# B&R Automation Studio project A_FullProject
Automation Studio 4.9

## Configuration Config1

CPU X20CP1686X, AutomationRuntime M4.93, Build 4.1.2, Safety 0.0, Vc V4.73.2

### Task classes (Cpu.sw)
```
Cyclic#4:
  Axis <- Vision.Axis.prg
  Vi_main <- Vision.Vi_main.prg
  Vi_image <- Vision.Vi_image.prg
DataObjects: McAcpSys
NcDataObjects: mcdrivelog
Binaries: arsvcreg, FWRules, McAcpSim, mvLoader, mCoWebSc, visionUnit, McAcpDrv, TCData, udbdef, arflatprv, arcoal, iomap, asfw, Settings, Role, SettingsVC, Config_1, VAMatch, arconfig, VCMyCam, ashwd, sysconf, User, ashwac
Libraries: McBase, MpBase, ViBase, AsZip, FileIO, AsARCfg, powerlnk, AsEPL, AsIO, AsTCP, sys_lib, DataObj, astime, runtime, CoTrace, MpAxis, McAxis, McAcpAx, arssl, asieccon
```

### Hardware
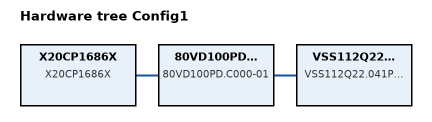
```
80VD100PD.C000-01 : 80VD100PD.C000-01 v2.5.0.0  [PLK1 -> X20CP1686X.IF3 (NodeNumber=1) [Cable Type=PowerlinkCable, Length=10, Version=1.0.0.3]; PLK2 -> VSS112Q22.041P-000.PLK1 (NodeNumber=1) [Cable Type=PowerlinkCable, Length=10, Version=1.0.0.3]]
  DriveConfiguration/Module:
    McAcoposTypeID = AcoposMicroDConfig
    ActivateACOPOSSimulationOnPLC = 0
  DriveConfiguration/Channel[1]/RealAxis:
    AxisReference = 
    MechanicalElementsIsInvisible = 0
  DriveConfiguration/Channel[1]/RealAxis/MechanicalElements/Gearbox:
    InputIsReadOnly = 0
    Input = 1
    OutputIsReadOnly = 0
    Output = 1
  DriveConfiguration/Channel[1]/RealAxis/MechanicalElements/RotaryToLinearTransformation:
    ReferenceDistanceIsReadOnly = 0
    ReferenceDistance = 1
  DriveConfiguration/Channel[1]/RealAxis/Controller:
    ModeIsReadOnly = 0
    Mode = PositionController
  DriveConfiguration/Channel[1]/RealAxis/Controller/Mode/Position:
    ProportionalGain = 200
    IntegrationTime = 0.0
    PredictionTime = 0.0004
    TotalDelayTime = 0.0004
  DriveConfiguration/Channel[1]/RealAxis/Controller/Mode/Speed:
    ProportionalGainIsReadOnly = 0
    ProportionalGain = 0.9
    IntegrationTimeIsReadOnly = 0
    IntegrationTime = 0.0
    FilterTimeIsReadOnly = 0
    FilterTime = 0.0
  DriveConfiguration/Channel[1]/RealAxis/Controller/Mode/LoopFilters:
    LoopFilterXIsReadOnly = 0
    LoopFilter1 = NotUsed
    LoopFilter2 = NotUsed
    LoopFilter3 = NotUsed
  DriveConfiguration/Channel[1]/RealAxis/Homing:
    ModeIsReadOnly = 0
    Mode = Direct
  DriveConfiguration/Channel[1]/RealAxis/Homing/Mode:
    Position = 0.0
    ReferencePulse = NotUsed
  DriveConfiguration/Channel[1]/RealAxis/Homing:
    RestorePositionVariable = 
  DriveConfiguration/Channel[1]/RealAxis/StopReaction:
    QuickstopIsReadOnly = 0
    Quickstop = DecelerationLimit
    DriveErrorIsReadOnly = 0
    DriveError = DecelerationLimit
  DriveConfiguration/Channel[1]/RealAxis/MovementErrorLimits:
    PositionError = 1.0
    VelocityErrorMonitoring = Automatic1
  DriveConfiguration/Channel[1]/RealAxis:
    JerkFilterIsReadOnly = 0
    JerkFilter = NotUsed
    ZeroVibrationFilter = NotUsed
  DriveConfiguration/Channel[1]/RealAxis/DigitalInputs/HomingSwitch:
    SourceIsReadOnly = 0
    Source = NotUsed
    Level = High
  DriveConfiguration/Channel[1]/RealAxis/DigitalInputs/PositiveLimitSwitch:
    SourceIsReadOnly = 0
    Source = NotUsed
    Level = High
  DriveConfiguration/Channel[1]/RealAxis/DigitalInputs/NegativeLimitSwitch:
    SourceIsReadOnly = 0
    Source = NotUsed
    Level = High
  DriveConfiguration/Channel[1]/RealAxis/DigitalInputs/Trigger1:
    Source = X2Trigger1
    Level = High
  DriveConfiguration/Channel[1]/RealAxis/DigitalInputs/Trigger2:
    Source = X2Trigger2
    Level = High
  DriveConfiguration/Channel[1]/RealAxis/DigitalInputs/Quickstop:
    Input = Trigger2
  DriveConfiguration/Channel[1]/RealAxis/Simulation:
    SimulationModeOnPLC = SetValueGeneration
    SimulationModeOnACOPOS = NotUsed
  DriveConfiguration/Channel[1]:
    ExternalEncoderAxis = NotUsed
  DriveConfiguration/Channel[2]/RealAxis:
    AxisReference = gAxis_1
    MechanicalElementsIsInvisible = 0
  DriveConfiguration/Channel[2]/RealAxis/MechanicalElements/Gearbox:
    InputIsReadOnly = 0
    Input = 1
    OutputIsReadOnly = 0
    Output = 1
  DriveConfiguration/Channel[2]/RealAxis/MechanicalElements/RotaryToLinearTransformation:
    ReferenceDistanceIsReadOnly = 0
    ReferenceDistance = 1
  DriveConfiguration/Channel[2]/RealAxis/Controller:
    ModeIsReadOnly = 0
    Mode = PositionController
  DriveConfiguration/Channel[2]/RealAxis/Controller/Mode/Position:
    ProportionalGain = 200
    IntegrationTime = 0.0
    PredictionTime = 0.0004
    TotalDelayTime = 0.0004
  DriveConfiguration/Channel[2]/RealAxis/Controller/Mode/Speed:
    ProportionalGainIsReadOnly = 0
    ProportionalGain = 0.9
    IntegrationTimeIsReadOnly = 0
    IntegrationTime = 0.0
    FilterTimeIsReadOnly = 0
    FilterTime = 0.0
  DriveConfiguration/Channel[2]/RealAxis/Controller/Mode/LoopFilters:
    LoopFilterXIsReadOnly = 0
    LoopFilter1 = NotUsed
    LoopFilter2 = NotUsed
    LoopFilter3 = NotUsed
  DriveConfiguration/Channel[2]/RealAxis/Homing:
    ModeIsReadOnly = 0
    Mode = Direct
  DriveConfiguration/Channel[2]/RealAxis/Homing/Mode:
    Position = 0.0
    ReferencePulse = NotUsed
  DriveConfiguration/Channel[2]/RealAxis/Homing:
    RestorePositionVariable = 
  DriveConfiguration/Channel[2]/RealAxis/StopReaction:
    QuickstopIsReadOnly = 0
    Quickstop = DecelerationLimit
    DriveErrorIsReadOnly = 0
    DriveError = DecelerationLimit
  DriveConfiguration/Channel[2]/RealAxis/MovementErrorLimits:
    PositionError = 1.0
    VelocityErrorMonitoring = Automatic1
  DriveConfiguration/Channel[2]/RealAxis:
    JerkFilterIsReadOnly = 0
    JerkFilter = NotUsed
    ZeroVibrationFilter = NotUsed
  DriveConfiguration/Channel[2]/RealAxis/DigitalInputs/HomingSwitch:
    SourceIsReadOnly = 0
    Source = NotUsed
    Level = High
  DriveConfiguration/Channel[2]/RealAxis/DigitalInputs/PositiveLimitSwitch:
    SourceIsReadOnly = 0
    Source = NotUsed
    Level = High
  DriveConfiguration/Channel[2]/RealAxis/DigitalInputs/NegativeLimitSwitch:
    SourceIsReadOnly = 0
    Source = NotUsed
    Level = High
  DriveConfiguration/Channel[2]/RealAxis/DigitalInputs/Trigger1:
    Source = X2Trigger1
    Level = High
  DriveConfiguration/Channel[2]/RealAxis/DigitalInputs/Trigger2:
    Source = X2Trigger2
    Level = High
  DriveConfiguration/Channel[2]/RealAxis/DigitalInputs/Quickstop:
    Input = Trigger2
  DriveConfiguration/Channel[2]/RealAxis/Simulation:
    SimulationModeOnPLC = SetValueGeneration
    SimulationModeOnACOPOS = NotUsed
  DriveConfiguration/Channel[2]:
    ExternalEncoderAxis = NotUsed
VSS112Q22.041P-000 : VSS112Q22.041P-000 v1.11.0.922  [PLK1 -> 80VD100PD.C000-01.PLK2 (NodeNumber=2) [Cable Type=PowerlinkCable, Length=10, Version=1.0.0.3]]
  Supervision = off
  VisionConfig = VCMyCam
X20CP1686X : X20CP1686X v1.8.2.0
  Connector IF2:
    ActivateDevice = 1
    Mode = Manual
    InternetAddress = 192.168.1.100
    SubnetMask = 255.255.255.0
    ActivateSnmp = 2
  Connector IF3:
    MtuSize = 1500
    InternetAddress = 192.168.200.240
    SubnetMask = 255.255.255.0
  ConfigurationID = VisionSample_AxisSync_Config1
  UserPartitionSize = 500
  TimerDeviceType = EPLX2X
  TimerDevice = X20CP1686X.IF3
  FileDevice1
  FileDeviceName1 = CF
  FileDevicePath1 = F:\
  FtpUser1
  FtpUsername1 = test
  FtpUserPassword1 = QkT+VSyJDE68GyHqQqfzGbDLRHfoQvgBAqgTYwFwErQ=  // test
  FtpUserSalt1 = 9xieoJwW
  FTPAccessRight1 = 0
  FTPdevice1 = ALL
  ActivateOpcUa = 1
  OpcUaInformationModels_PV_Version = 1
```

### IoMap.iom - X20CP1686X/IoMap.iom
```iecst
VAR_CONFIG
	::Vi_main:VisionCtrl.Parameters.SetFocus AT %QW."VSS112Q22.041P-000".SetFocus;
	::Vi_main:VisionCtrl.Parameters.ExposureTime AT %QD."VSS112Q22.041P-000".ExposureTime01;
	::Vi_main:VisionCtrl.Parameters.FlashColor AT %QB."VSS112Q22.041P-000".FlashColor01;
	::Vi_main:VisionCtrl.Parameters.FlashSegment AT %QB."VSS112Q22.041P-000".FlashSegment01;
	::Vi_main:CompletedAcquisitionCntOld AT %IB."VSS112Q22.041P-000".CompletedAcquisitionCnt;
END_VAR
```

### Config_1.axis - X20CP1686X/mappMotion/Config_1.axis
```
Element gAxis_1 (Type=axis)
  BaseTypeIsReadOnly = 0
  BaseType = RotaryPeriodic
    MeasurementUnitIsReadOnly = 0
    MeasurementUnit = 17476
    MeasurementResolutionIsReadOnly = 0
    MeasurementResolution = 0.01
    CountDirectionIsReadOnly = 0
    CountDirection = Standard
    PeriodSettings:
      Period = 360.0
  MovementLimitsIsReadOnly = 0
  MovementLimits = Internal
    Position:
      LowerLimitMin = -1.79769313486231E308
      UpperLimitMax = 1.79769313486231E308
      LowerLimit = -1000.0
      UpperLimit = 1000.0
    VelocityIsReadOnly = 0
    Velocity:
      VelocityMax = 3.4E38
      Velocity = 6000
    AccelerationIsReadOnly = 0
    Acceleration:
      AccelerationMax = 3.4E38
      Acceleration = 36000
    DecelerationIsReadOnly = 0
    Deceleration:
      DecelerationMax = 3.4E38
      Deceleration = 36000
  Alarms = None
```

### SettingsVC.vicfg - X20CP1686X/mappVision/SettingsVC.vicfg
```
Element VisionSettings (Type=vicfg)
  ActivateVisualization = TRUE
  FileDeviceName
  Permissions:
    WriteAccessRole = Everyone
  DeepLearning:
    CustomDlNetworks:
      DLFileDeviceName
      DLNetworkBuildPath
```

### VCMyCam.visioncomponent - X20CP1686X/mappVision/VCMyCam.visioncomponent
```
Element VCMyCam (Type=visioncomponent)
  VisionApplicationReference = VAMatch
```

## Logical view

Binary libraries used (declarations not repeated): brsystem, McAcpAx 5.28.2, McBase 5.28.2, powerlnk, ViBase 5.28.1

### Package Logical/Libraries - Globale Bibliotheken

### MpAxisCfg.typ
```iecst
TYPE
	MpAXBAxBaseTypEnum :
		( (*Axis base type*)
		mcAXB_BASE_TYPE_LIN_BD := 0, (*Linear bounded - Linear axis with bounded movement scope*)
		mcAXB_BASE_TYPE_LIN := 1, (*Linear - Linear axis*)
		mcAXB_BASE_TYPE_LIN_PER := 2, (*Linear periodic - Linear axis with periodic movement scope*)
		mcAXB_BASE_TYPE_ROT_BD := 10, (*Rotary bounded - Rotary axis with bounded movement scope*)
		mcAXB_BASE_TYPE_ROT := 11, (*Rotary - Rotary axis*)
		mcAXB_BASE_TYPE_ROT_PER := 12 (*Rotary periodic - Rotary axis with periodic movement scope*)
		);
	MpAXBAxMeasUnitEnum :
		( (*Measurement unit for the axis*)
		mcAXB_MEAS_UNIT_G_SET := 0, (*Global settings*)
		mcAXB_MEAS_UNIT_MILIMETERS := 5066068, (*Milimeters*)
		mcAXB_MEAS_UNIT_M := 5067858, (*Meters*)
		mcAXB_MEAS_UNIT_INCH := 4804168, (*Inches*)
		mcAXB_MEAS_UNIT_DEG := 17476, (*Degrees*)
		mcAXB_MEAS_UNIT_GRAD := 4274481, (*Gradians*)
		mcAXB_MEAS_UNIT_REV := 5059636, (*Revolutions*)
		mcAXB_MEAS_UNIT_GEN := -1 (*Generic*)
		);
	MpAXBAxCntDirEnum :
		( (*Direction of the axis in which the position value is increasing*)
		mcAXB_COUNT_DIR_STD := 0, (*Standard*)
		mcAXB_COUNT_DIR_INV := 1 (*Inverse*)
		);
	MpAXBAxMoveLimTypEnum :
		( (*Movement limits settings*)
		mcAXB_MOV_LIM_STD := 0, (*Standard*)
		mcAXB_MOV_LIM_PATH_CTRL_AX := 1, (*Path controlled axis*)
		mcAXB_MOV_LIM_LIM_SET_REF := 2 (*Limit set reference*)
		);
	MpAXBAxMoveLimPosType : STRUCT (*Movement range of the axis via two position boundaries; Only for bounded axis*)
		LowerLimit : LREAL; (*Lower software limit position [Measurement units]*)
		UpperLimit : LREAL; (*Upper software limit position [Measurement units]*)
	END_STRUCT;
	MpAXBAxMoveLimVelType : STRUCT (*Limits for the velocity of the axis*)
		Positive : REAL; (*Velocity limit in positive movement direction [Measurement units/s]*)
		Negative : REAL; (*Velocity limit in negative movement direction [Measurement units/s]*)
	END_STRUCT;
	MpAXBAxMoveLimType : STRUCT
		Type : MpAXBAxMoveLimTypEnum; (*Movement limits settings*)
		Position : MpAXBAxMoveLimPosType; (*Movement range of the axis via two position boundaries; Only for bounded axis*)
		Velocity : MpAXBAxMoveLimVelType; (*Limits for the velocity of the axis*)
		Acceleration : REAL; (*Acceleration limit in any movement direction [Measurement units/s²]*)
		Deceleration : REAL; (*Deceleration limit in any movement direction [Measurement units/s²]*)
		Jerk : REAL; (*Jerk limit in any movement direction [Measurement units/s³]; Only for [Measurement units/s³]*)
		Torque : REAL; (*Torque limit in any movement direction; Only for Axis of type rotary; only for limits type internal path controlled [Nm]*)
		Force : REAL; (*Force limit in any movement direction [N]; Only for Axis of type linear; only for limits type internal path controlled [N]*)
		LimitSetReference : STRING[250]; (*Name of the limit reference; only for limits type external*)
	END_STRUCT;
	MpAXBAxType : STRUCT (*Axis configuration*)
		BaseType : MpAXBAxBaseTypEnum; (*Axis base type*)
		MeasurementUnit : MpAXBAxMeasUnitEnum; (*Measurement unit for the axis*)
		MeasurementResolution : LREAL; (*Possible resolution of measurement unit that can be achieved [Measurement resolution]*)
		CountDirection : MpAXBAxCntDirEnum; (*Direction of the axis in which the position value is increasing*)
		Period : LREAL; (*The value range for axis positions is [0 , Period]; Only for Axis of type periodic [Measurement units]*)
		MovementLimits : MpAXBAxMoveLimType;
	END_STRUCT;
	MpAXBDrvMechElmGBType : STRUCT
		Input : DINT; (*Number of rotations on the encoder side [Revolutions] [Revolutions]*)
		Output : DINT; (*Number of rotations on the load side which correspond to the number of rotations onthe encoder side [Revolutions] [Revolutions]*)
	END_STRUCT;
	MpAXBDrvMechElmRotToLinTrfType : STRUCT (*Specifies a transformation factor between the output of the gear and the actual load movement*)
		ReferenceDistance : LREAL; (*Reference distance which is considered for an axis positioning [Measurement units/Gearbox output revolution] [Measurement units/Gearbox output revolution]*)
	END_STRUCT;
	MpAXBDrvMechElmType : STRUCT (*Parameter of hardware elements situated between motor encoder and load which influence the scaling*)
		Gearbox : MpAXBDrvMechElmGBType;
		RotaryToLinearTransformation : MpAXBDrvMechElmRotToLinTrfType; (*Specifies a transformation factor between the output of the gear and the actual load movement*)
	END_STRUCT;
	MpAXBDrvCtrlModEnum :
		( (*Mode of the axis controller*)
		mcAXB_CTRL_MODE_POS := 0, (*Position - Automatic speed feed-forward with prediction time > 0*)
		mcAXB_CTRL_MODE_POS_W_TORQ_FF := 1, (*Position with torque FF - Torque feed-forward with specified parameters*)
		mcAXB_CTRL_MODE_POS_MDL_BASED := 3, (*Position model based - Model based control with specified parameters*)
		mcAXB_CTRL_MODE_V_FREQ := 2, (*Voltage frequency - Voltage/frequency control of induction motor with specified parameters*)
		mcAXB_CTRL_MODE_STP_CUR := 4, (*Stepper current - StpAx only. Current controller is used*)
		mcAXB_CTRL_MODE_STP_POS_AND_CUR := 5, (*Stepper position and current - StpAx only. Position and current controller are used*)
		mcAXB_CTRL_MODE_NOT_USE := 6 (*Not used - Controller not used*)
		);
	MpAXBDrvCtrlPosType : STRUCT (*Position controller parameters*)
		ProportionalGain : REAL; (*Proportional amplification [1/s]*)
		IntegrationTime : REAL; (*Integral action time [s]*)
		TotalDelayTime : REAL; (*Total delay time [s]*)
		PredictionTime : REAL; (*Prediction time [s]*)
		MaximumProportionalAction : REAL; (*Maximum proportional action. Only for StpAx and PureVax with GPAI [Measurement units/s]*)
		MaximumIntegralAction : REAL; (*Maximum integral action. Only for PureVax with GPAI [Measurement units/s]*)
	END_STRUCT;
	MpAXBDrvCtrlSpdType : STRUCT (*Speed controller parameters*)
		ProportionalGain : REAL; (*Proportional amplification [1/s]*)
		IntegrationTime : REAL; (*Integral action time [s]*)
		FilterTime : REAL; (*Filter time constant [s]*)
	END_STRUCT;
	MpAXBDrvCtrlFFwdModEnum :
		( (*Mode of the axis controller*)
		mcAXB_FF_MODE_STD := 0, (*Standard*)
		mcAXB_FF_MODE_PRED_SPD := 1, (*Predictive speed*)
		mcAXB_FF_MODE_TWO_MASS_MDL := 2 (*Two mass model*)
		);
	MpAXBDrvCtrlFFwdType : STRUCT (*Torque feed-forward control parameters*)
		Mode : MpAXBDrvCtrlFFwdModEnum; (*Mode of the axis controller*)
		TorqueLoad : REAL; (*Load torque [Nm]*)
		TorquePositive : REAL; (*Torque in positive direction [Nm]*)
		TorqueNegative : REAL; (*Torque in negative direction [Nm]*)
		SpeedTorqueFactor : REAL; (*Speed torque factor [Nms]*)
		Inertia : REAL; (*Mass moment of inertia [kgm²]*)
		AccelerationFilterTime : REAL; (*Acceleration filter time constant [s]*)
		PredictionTime : REAL; (*Prediction time [s]*)
	END_STRUCT;
	MpAXBDrvCtrlFdbkModEnum :
		( (*Mode of the axis controller*)
		mcAXB_CTLR_FEED_STD := 0, (*Standard*)
		mcAXB_CTLR_FEED_ONE_MASS_MDL := 1, (*One mass model*)
		mcAXB_CTLR_FEED_TWO_MASS_MDL := 2, (*Two mass model*)
		mcAXB_CTLR_FEED_TWO_ENC_SPD := 3 (*Two encoder speed*)
		);
	MpAXBDrvCtrlFdbkType : STRUCT (*Feedback control parameters*)
		Mode : MpAXBDrvCtrlFdbkModEnum; (*Mode of the axis controller*)
		SpeedMixingFactor : REAL; (*Load torque [Nm]*)
		SpeedProportionalGain : REAL; (*Torque in positive direction [Nm]*)
	END_STRUCT;
	MpAXBDrvCtrlMdlMass1Type : STRUCT (*Mass 1 parameters*)
		Inertia : REAL; (*Mass moment of inertia [kgm²]*)
		ViscousFriction : REAL; (*Viscous friction [Nms]*)
	END_STRUCT;
	MpAXBDrvCtrlMdlMass2Type : STRUCT (*Mass 2 parameters*)
		Inertia : REAL; (*Mass moment of inertia [kgm²]*)
		ViscousFriction : REAL; (*Viscous friction [Nms]*)
		Stiffness : REAL; (*Stiffness of the coupling to mass 1 [Nm/rad]*)
		Damping : REAL; (*Damping of the coupling to mass 1 [Nms/rad]*)
	END_STRUCT;
	MpAXBDrvCtrlMdlType : STRUCT (*Load model parameters*)
		Mass1 : MpAXBDrvCtrlMdlMass1Type; (*Mass 1 parameters*)
		Mass2 : MpAXBDrvCtrlMdlMass2Type; (*Mass 2 parameters*)
	END_STRUCT;
	MpAXBDrvCtrlVFreqCtrlTypEnum :
		( (*Type of characteristic curve*)
		mcAXB_VF_TYP_LIN := 129, (*Linear - Linear characteristic curve*)
		mcAXB_VF_TYP_CONST_LD_TORQ := 131, (*Constant load torque - Characteristic curve for quadratic load curves*)
		mcAXB_VF_TYP_QUAD := 130 (*Quadratic - Characteristic curve for quadratic load curves*)
		);
	MpAXBDrvCtrlVFreqCtrlAutCfgEnum :
		( (*Automatic configuration of parameters*)
		mcAXB_VF_AUTO_CFG_NOT_USE := 0, (*Not used*)
		mcAXB_VF_AUTO_CFG_MOT_PAR_BASED := 1 (*Motor parameter based*)
		);
	MpAXBDrvCtrlVFreqCtrlType : STRUCT (*V/f control parameters*)
		Type : MpAXBDrvCtrlVFreqCtrlTypEnum; (*Type of characteristic curve*)
		AutomaticConfiguration : MpAXBDrvCtrlVFreqCtrlAutCfgEnum; (*Automatic configuration of parameters*)
		SlipCompensation : REAL; (*Slip compensation: Multiplication factor of compensated frequency*)
		TotalDelayTime : REAL; (*Total delay time [s]*)
		BoostVoltage : REAL; (*Boost voltage [V]*)
		RatedVoltage : REAL; (*Rated voltage [V]*)
		RatedFrequency : REAL; (*Rated frequency [cps]*)
	END_STRUCT;
	MpAXBDrvCtrlLoopFltrTypEnum :
		( (*Type of the loop filter*)
		mcAXB_LP_FLTR_NOT_USE := 0, (*Not used - Filter is not active*)
		mcAXB_LP_FLTR_LOW_PASS_2ND_ORD := 1, (*Low pass 2nd order*)
		mcAXB_LP_FLTR_NOTCH := 2, (*Notch*)
		mcAXB_LP_FLTR_BIQUAD := 3, (*Biquad*)
		mcAXB_LP_FLTR_DISC_TIME_TRAN_FUN := 4, (*Discrete time transfer function*)
		mcAXB_LP_FLTR_LIM := 5, (*Limiter*)
		mcAXB_LP_FLTR_LIN_LIM := 6, (*Linear limitation*)
		mcAXB_LP_FLTR_RISE_TIME_LIM := 7, (*Rise time limitation*)
		mcAXB_LP_FLTR_COMP := 8 (*Compensation*)
		);
	MpAXBLoopFltrLP2ndOrdType : STRUCT (*Lowpass 2nd order*)
		CutOffFrequency : REAL; (*Cut off frequency [Hz]*)
	END_STRUCT;
	MpAXBLoopFltrNotchType : STRUCT (*Notch*)
		CenterFrequency : REAL; (*Center frequency [Hz]*)
		Bandwidth : REAL; (*Bandwidth [Hz]*)
	END_STRUCT;
	MpAXBLoopFltrBiquadType : STRUCT (*Biquad*)
		FrequencyNumerator : REAL; (*Frequency numerator [Hz]*)
		DampingNumerator : REAL; (*Damping numerator*)
		FrequencyDenominator : REAL; (*Frequency denominator [Hz]*)
		DampingDenominator : REAL; (*Damping Denominator*)
	END_STRUCT;
	MpAXBLoopFltrDiscTimeTranFunType : STRUCT (*Discrete time transfer function*)
		CoeffA0DenominatorPolynomial : REAL; (*Coefficient a0 of denominator polynomial*)
		CoeffA1DenominatorPolynomial : REAL; (*Coefficient a1 of denominator polynomial*)
		CoeffB0NominatorPolynomial : REAL; (*Coefficient b0 of numerator polynomial*)
		CoeffB1NominatorPolynomial : REAL; (*Coefficient b1 of numerator polynomial*)
		CoeffB2NominatorPolynomial : REAL; (*Coefficient b2 of numerator polynomial*)
	END_STRUCT;
	MpAXBLoopFltrLimLimTypEnum :
		( (*Select if for the limit a fixed value or if the value of an ACOPOS ParID is used*)
		mcAXB_LOOP_FLTR_LIM_TYPE_PARID := 0, (*ParId*)
		mcAXB_LOOP_FLTR_LIM_TYPE_FIX_VAL := 1 (*Fixed value*)
		);
	MpAXBLoopFltrLimLimType : STRUCT (*Positive limit setting*)
		Type : MpAXBLoopFltrLimLimTypEnum; (*Select if for the limit a fixed value or if the value of an ACOPOS ParID is used*)
		ParID : UINT; (*ParID*)
		Value : REAL; (*Value [A]*)
	END_STRUCT;
	MpAXBLoopFltrLimType : STRUCT (*Limiter*)
		PositiveLimit : MpAXBLoopFltrLimLimType; (*Positive limit setting*)
		NegativeLimit : MpAXBLoopFltrLimLimType; (*Negative limit setting*)
	END_STRUCT;
	MpAXBLoopFltrLinLimType : STRUCT (*Linear limitation*)
		InputParID : UINT; (*ACOPOS ParID for the input*)
		InputLimit : REAL; (*Input limit value for full limitation*)
		Gradient : REAL; (*Gradient*)
	END_STRUCT;
	MpAXBLoopFltrRiseTimeLimType : STRUCT (*Rise time limitation*)
		RiseTime : REAL; (*Rise time [s]*)
		NormalizedLimit : REAL; (*Normalized limit*)
	END_STRUCT;
	MpAXBLoopFltrCompType : STRUCT (*Compensation*)
		MultiplicationFactorParID : UINT; (*Multiplication Factor ParID*)
		AdditiveValueParID : UINT; (*Additive Value ParID*)
	END_STRUCT;
	MpAXBDrvCtrlLoopFltrLoopFltrType : STRUCT (*Type of the loop filter*)
		Type : MpAXBDrvCtrlLoopFltrTypEnum; (*Type of the loop filter*)
		Lowpass2ndOrder : MpAXBLoopFltrLP2ndOrdType; (*Lowpass 2nd order*)
		Notch : MpAXBLoopFltrNotchType; (*Notch*)
		Biquad : MpAXBLoopFltrBiquadType; (*Biquad*)
		DiscreteTimeTransferFunction : MpAXBLoopFltrDiscTimeTranFunType; (*Discrete time transfer function*)
		Limiter : MpAXBLoopFltrLimType; (*Limiter*)
		LinearLimitation : MpAXBLoopFltrLinLimType; (*Linear limitation*)
		RiseTimeLimitation : MpAXBLoopFltrRiseTimeLimType; (*Rise time limitation*)
		Compensation : MpAXBLoopFltrCompType; (*Compensation*)
	END_STRUCT;
	MpAXBDrvCtrlLoopFltrType : STRUCT (*Parameters of the loop filters*)
		LoopFilter : ARRAY[0..2] OF MpAXBDrvCtrlLoopFltrLoopFltrType; (*Type of the loop filter*)
	END_STRUCT;
	MpAXBDrvCtrlCurModEnum :
		( (*Mode of current controller*)
		mcAXB_CUR_CTRL_MODE_STD := 0 (*Standard*)
		);
	MpAXBDrvCtrlCurType : STRUCT (*Current controller parameters; Only for stepper axis*)
		Mode : MpAXBDrvCtrlCurModEnum; (*Mode of current controller*)
		StandstillCurrent : REAL; (*Current that is used when no movement is active [A]*)
		ConstantSpeedCurrent : REAL; (*Current that is used when a movement with a constant speed is active [A]*)
		SpeedChangeCurrent : REAL; (*Current that is used when the axis is accelerating or decelerating [A]*)
		FullStepThreshold : REAL; (*Speed of the motor where the driver switch from microstep to full step mode [rpm]*)
		MotorSettlingTime : REAL; (*Minimum time between when the motor is powered on to when the DrvOk bit is set. Settings made in steps of 10 ms. [s]*)
		DelayedCurrentSwitchOff : REAL; (*Time for a delayed motor switch off after it is decelerated to zero because of a settime fault. Setting is made in steps of 100 ms. [s]*)
	END_STRUCT;
	MpAXBDrvCtrlType : STRUCT (*Axis controller parameters*)
		Mode : MpAXBDrvCtrlModEnum; (*Mode of the axis controller*)
		Position : MpAXBDrvCtrlPosType; (*Position controller parameters*)
		Speed : MpAXBDrvCtrlSpdType; (*Speed controller parameters*)
		FeedForward : MpAXBDrvCtrlFFwdType; (*Torque feed-forward control parameters*)
		Feedback : MpAXBDrvCtrlFdbkType; (*Feedback control parameters*)
		Model : MpAXBDrvCtrlMdlType; (*Load model parameters*)
		VoltageFrequencyControl : MpAXBDrvCtrlVFreqCtrlType; (*V/f control parameters*)
		LoopFilters : MpAXBDrvCtrlLoopFltrType; (*Parameters of the loop filters*)
		Current : MpAXBDrvCtrlCurType; (*Current controller parameters; Only for stepper axis*)
	END_STRUCT;
	MpAXBDrvHomeType : STRUCT (*Homing mode and parameters which can be used within the application program as pre-configured setting*)
		Mode : McHomingModeEnum; (*Mode of the axis controller*)
		Position : LREAL; (*Home position [Measurement units]*)
		ReferencePulse : McSwitchEnum; (*Use reference pulse of encoder*)
		ReferencePulseBlockingDistance : LREAL; (*Distance for blocking the activation of triggering reference pulse [Measurement units]*)
		StartVelocity : REAL; (*Speed for searching the reference switch [Measurement units/s]*)
		HomingVelocity : REAL; (*Speed which is used while searching for the homing event (e.g. after reference switch has been reached) [Measurement units/s]*)
		Acceleration : REAL; (*Acceleration for homing movement [Measurement units/s²]*)
		SwitchEdge : McDirectionEnum; (*Edge of reference switch*)
		HomingDirection : McDirectionEnum; (*Movement direction in which the homing event is evaluated*)
		StartDirection : McDirectionEnum; (*Start direction of movement for searching the reference*)
		KeepDirection : McSwitchEnum; (*Keep direction (move only in one direction)*)
		TorqueLimit : REAL; (*Torque limit for homing on block [Nm]*)
		PositionErrorStopLimit : LREAL; (*Lag error for stop of the homing movement [Measurement units/s²]*)
		BlockDetectionPositionError : LREAL; (*Lag error for block detection [Measurement units]*)
		RestorePositionVariable : STRING[250]; (*Remanent variable used for homing mode: Restore position*)
	END_STRUCT;
	MpAXBDrvStopReacQstopEnum :
		( (*Reaction in case of a quickstop which is caused by an active quickstop input*)
		mcAXB_QSTOP_RCT_DEC_LIM := 0, (*Deceleration limit*)
		mcAXB_QSTOP_RCT_DEC_LIM_W_JERK := 1, (*Deceleration limit with jerk*)
		mcAXB_QSTOP_RCT_TORQ_LIM := 2, (*Torque limit*)
		mcAXB_QSTOP_RCT_INDUCT_HALT := 3 (*Induction halt*)
		);
	MpAXBDrvStopReacDrvErrEnum :
		( (*Reaction in case of an error stop which is caused by a drive error*)
		mcAXB_ERR_RCT_DEC_LIM := 0, (*Deceleration limit*)
		mcAXB_ERR_RCT_INDUCT_HALT := 1, (*Induction halt*)
		mcAXB_ERR_RCT_COAST_STANDSTILL := 2, (*Coast standstill*)
		mcAXB_ERR_RCT_CYC_DEC_AXESGROUP := 3 (*Cyclic deceleration AxesGroup*)
		);
	MpAXBDrvStopReacType : STRUCT (*Reactions of the axis in case of certain stop conditions*)
		Quickstop : MpAXBDrvStopReacQstopEnum; (*Reaction in case of a quickstop which is caused by an active quickstop input*)
		DriveError : MpAXBDrvStopReacDrvErrEnum; (*Reaction in case of an error stop which is caused by a drive error*)
	END_STRUCT;
	MpAXBDrvMovVelErrMonEnum :
		( (*Velocity error monitoring mode*)
		mcAXB_VEL_MON_AUT_1 := 0, (*Automatic 1*)
		mcAXB_VEL_MON_AUT_2 := 1, (*Automatic 2*)
		mcAXB_VEL_MON_USR_DEF := 2, (*User defined*)
		mcAXB_VEL_MON_NOT_USE := 3 (*Not used*)
		);
	MpAXBDrvMovementErrorLimitsType : STRUCT (*Limit values that result in a stop reaction when exceeded*)
		PositionError : LREAL; (*Lag error limit for stopping a movement [Measurement units]*)
		VelocityErrorMonitoring : MpAXBDrvMovVelErrMonEnum; (*Velocity error monitoring mode*)
		VelocityError : REAL; (*Velocity error limit for stopping a movement [Measurement units/s]*)
	END_STRUCT;
	MpAXBDrvJerkFilterTypEnum :
		( (*Jerk filter setting*)
		mcAXB_JERK_FLTR_NOT_USE := 0, (*Not used*)
		mcAXB_JERK_FLTR_TIME := 1, (*Time*)
		mcAXB_JERK_FLTR_LIM := 2 (*Limited*)
		);
	MpAXBDrvJerkFilterType : STRUCT (*Jerk filter*)
		Type : MpAXBDrvJerkFilterTypEnum; (*Jerk filter setting*)
		Jerk : REAL; (*Dependant on selected type it is either the jerk limit in any movement direction or a jerk filter time.*)
	END_STRUCT;
	MpAXBDrvDigInLevelEnum :
		( (*Level of the digital input hardware which leads to an active level of the functionality*)
		mcAXB_DI_LEVEL_HIGH := 0, (*High*)
		mcAXB_DI_LEVEL_LOW := 1 (*Low*)
		);
	MpAXBDrvDigInSrcEnum :
		( (*Source of the digital input which is used for this functionality*)
		mcAXBDI_NOT_USE := 0, (*Not used*)
		mcAXBDI_ACP_DIG_IN_X8TRG_1 := 1, (*ACOPOS digital in X8.Trigger 1*)
		mcAXBDI_ACP_DIG_IN_X8TRG_2 := 2, (*ACOPOS digital in X8.Trigger 2*)
		mcAXBDI_ACP_DIG_IN_SS1X41X1 := 3, (*ACOPOS digital in SS1.X41x.1*)
		mcAXBDI_ACP_DIG_IN_SS1X41X2 := 4, (*ACOPOS digital in SS1.X41x.2*)
		mcAXBDI_ACP_DIG_IN_SS1X41X3 := 5, (*ACOPOS digital in SS1.X41x.3*)
		mcAXBDI_ACP_DIG_IN_SS1X41X4 := 6, (*ACOPOS digital in SS1.X41x.4*)
		mcAXBDI_ACP_DIG_IN_SS1X41X5 := 7, (*ACOPOS digital in SS1.X41x.5*)
		mcAXBDI_ACP_DIG_IN_SS1X41X6 := 8, (*ACOPOS digital in SS1.X41x.6*)
		mcAXBDI_ACP_DIG_IN_SS1X41X7 := 9, (*ACOPOS digital in SS1.X41x.7*)
		mcAXBDI_ACP_DIG_IN_SS1X41X8 := 10, (*ACOPOS digital in SS1.X41x.8*)
		mcAXBDI_ACP_DIG_IN_SS1X41X9 := 11, (*ACOPOS digital in SS1.X41x.9*)
		mcAXBDI_ACP_DIG_IN_SS1X41X10 := 12, (*ACOPOS digital in SS1.X41x.10*)
		mcAXBDI_ACP_DIG_IN_X23ATRG_1 := 13, (*ACOPOS digital in X23A.Trigger 1*)
		mcAXBDI_ACP_DIG_IN_X23ATRG_2 := 14, (*ACOPOS digital in X23A.Trigger 2*)
		mcAXBDI_ACP_DIG_IN_X24ATRG_2 := 15, (*ACOPOS digital in X24A.Trigger 2*)
		mcAXBDI_ACP_DIG_IN_X2TRG_1 := 16, (*ACOPOS digital in X2.Trigger 1*)
		mcAXBDI_ACP_DIG_IN_X2TRG_2 := 17, (*ACOPOS digital in X2.Trigger 2*)
		mcAXBDI_ACP_DIG_IN_X1TRG_1 := 18, (*ACOPOS digital in X1.Trigger 1*)
		mcAXBDI_ACP_DIG_IN_X1TRG_2 := 19, (*ACOPOS digital in X1.Trigger 2*)
		mcAXBDI_ACP_DIG_IN_X1REF_SW := 20, (*ACOPOS digital in X1.Reference switch*)
		mcAXBDI_ACP_DIG_IN_X1POS_HW_LIM := 21, (*ACOPOS digital in X1.Positive HW limit*)
		mcAXBDI_ACP_DIG_IN_X1NEG_HW_LIM := 22, (*ACOPOS digital in X1.Negative HW limit*)
		mcAXBDI_FORCED_BY_FUN_BLK := 23, (*Forced by function block*)
		mcAXBDI_VAR := 24, (*Variable*)
		mcAXBDI_IO_CH := 40, (*I/O Channel*)
		mcAXBDI_STP_DIG_IN_TRG_1 := 41, (*Stepper digital input trigger 1*)
		mcAXBDI_STP_DIG_IN_TRG_2 := 42, (*Stepper digital input trigger 2*)
		mcAXBDI_STP_DIG_IN_1 := 43, (*Stepper digital input 1*)
		mcAXBDI_STP_DIG_IN_2 := 44, (*Stepper digital input 2*)
		mcAXBDI_STP_DIG_IN_3 := 45, (*Stepper digital input 3*)
		mcAXBDI_STP_DIG_IN_4 := 46, (*Stepper digital input 4*)
		mcAXBDI_STP_DIG_IN_5 := 47, (*Stepper digital input 5*)
		mcAXBDI_STP_DIG_IN_6 := 48 (*Stepper digital input 6*)
		);
	MpAXBDrvDigInHomeSwType : STRUCT (*Homing switch input functionality*)
		Level : MpAXBDrvDigInLevelEnum; (*Level of the digital input hardware which leads to an active level of the functionality*)
		Source : MpAXBDrvDigInSrcEnum; (*Source of the digital input which is used for this functionality*)
		SourceMapping : STRING[250]; (*Process variable or IO channel source for digital input when type mcAXBDI_VAR or mcAXBDI_IO_CH is used*)
	END_STRUCT;
	MpAXBDrvDigInPosLimSwType : STRUCT (*Positive limit switch input functionality*)
		Level : MpAXBDrvDigInLevelEnum; (*Level of the digital input hardware which leads to an active level of the functionality*)
		Source : MpAXBDrvDigInSrcEnum; (*Source of the digital input which is used for this functionality*)
		SourceMapping : STRING[250]; (*Process variable or IO channel source for digital input when type mcAXBDI_VAR or mcAXBDI_IO_CH is used*)
	END_STRUCT;
	MpAXBDrvDigInNegLimSwType : STRUCT (*Negative limit switch input functionality*)
		Level : MpAXBDrvDigInLevelEnum; (*Level of the digital input hardware which leads to an active level of the functionality*)
		Source : MpAXBDrvDigInSrcEnum; (*Source of the digital input which is used for this functionality*)
		SourceMapping : STRING[250]; (*Process variable or IO channel source for digital input when type mcAXBDI_VAR or mcAXBDI_IO_CH is used*)
	END_STRUCT;
	MpAXBDrvDigTimeStampTypeEnum :
		( (*Time stamp setting*)
		mcAXB_DI_TIME_STAMP_NOT_USE := 0, (*Not used*)
		mcAXB_DI_TIME_STAMP_USE := 1, (*Used*)
		mcAXB_DI_TIME_STAMP_RIS_FALL_EDG := 2 (*Rising falling edge*)
		);
	MpAXBDrvDigTimeStampEdgType : STRUCT (*Parameters for the rising trigger edge for type mcAXB_DI_TIME_STAMP_RIS_FALL_EDG*)
		CountSourceMapping : STRING[250]; (*Name of the process variable (SINT) representing the trigger edge count*)
		TimeStampSourceMapping : STRING[250]; (*Name of the process variable (INT) representing the trigger edge time*)
	END_STRUCT;
	MpAXBDrvDigTimeStampType : STRUCT (*Trigger time stamp. StpAx only*)
		Type : MpAXBDrvDigTimeStampTypeEnum; (*Time stamp setting*)
		TimeStampSourceMapping : STRING[250]; (*Process variable time stamp source PV mapping for type mcAXB_DI_TIME_STAMP_USE*)
		RisingEdge : MpAXBDrvDigTimeStampEdgType; (*Parameters for the rising trigger edge for type mcAXB_DI_TIME_STAMP_RIS_FALL_EDG*)
		FallingEdge : MpAXBDrvDigTimeStampEdgType; (*Parameters for the falling trigger edge for type mcAXB_DI_TIME_STAMP_RIS_FALL_EDG*)
	END_STRUCT;
	MpAXBDrvDigInTrg1Type : STRUCT (*Trigger 1 input functionality*)
		Level : MpAXBDrvDigInLevelEnum; (*Level of the digital input hardware which leads to an active level of the functionality*)
		Source : MpAXBDrvDigInSrcEnum; (*Source of the digital input which is used for this functionality*)
		SourceMapping : STRING[250]; (*Process variable or IO channel source for digital input when type mcAXBDI_VAR or mcAXBDI_IO_CH is used*)
		TimeStamp : MpAXBDrvDigTimeStampType; (*Trigger time stamp. StpAx only*)
	END_STRUCT;
	MpAXBDrvDigInTrg2Type : STRUCT (*Trigger 2 input functionality*)
		Level : MpAXBDrvDigInLevelEnum; (*Level of the digital input hardware which leads to an active level of the functionality*)
		Source : MpAXBDrvDigInSrcEnum; (*Source of the digital input which is used for this functionality*)
		SourceMapping : STRING[250]; (*Process variable or IO channel source for digital input when type mcAXBDI_VAR or mcAXBDI_IO_CH is used*)
		TimeStamp : MpAXBDrvDigTimeStampType; (*Trigger time stamp. StpAx only*)
	END_STRUCT;
	MpAXBDrvDigInQstopInEnum :
		( (*Digital input functionality triggering an axis quickstop*)
		mcAXB_QSTOP_IN_TRG_2 := 0, (*Trigger 2*)
		mcAXB_QSTOP_IN_TRG_1 := 1, (*Trigger 1*)
		mcAXB_QSTOP_IN_POS_LIM_SW := 2, (*Positive limit switch*)
		mcAXB_QSTOP_IN_NEG_LIM_SW := 3, (*Negative limit switch*)
		mcAXB_QSTOP_IN_HOME_SW := 4, (*Homing switch*)
		mcAXB_QSTOP_IN_NOT_USE := 5, (*Not used*)
		mcAXB_QSTOP_IN_VAR := 6, (*Variable*)
		mcAXB_QSTOP_IN_IO_CH := 7 (*I/O Channel*)
		);
	MpAXBDrvDigInQstopType : STRUCT (*Quickstop input functionality*)
		Input : MpAXBDrvDigInQstopInEnum; (*Digital input functionality triggering an axis quickstop*)
		SourceMapping : STRING[250]; (*Process variable or IO channel source for digital input when following inputs types are used: mcAXB_QSTOP_VAR, mcAXB_QSTOP_IO_CH*)
	END_STRUCT;
	MpAXBDrvDigInType : STRUCT (*Various digital input functionalities e.g. like homing switch or triggers*)
		HomingSwitch : MpAXBDrvDigInHomeSwType; (*Homing switch input functionality*)
		PositiveLimitSwitch : MpAXBDrvDigInPosLimSwType; (*Positive limit switch input functionality*)
		NegativeLimitSwitch : MpAXBDrvDigInNegLimSwType; (*Negative limit switch input functionality*)
		Trigger1 : MpAXBDrvDigInTrg1Type; (*Trigger 1 input functionality*)
		Trigger2 : MpAXBDrvDigInTrg2Type; (*Trigger 2 input functionality*)
		Quickstop : MpAXBDrvDigInQstopType; (*Quickstop input functionality*)
	END_STRUCT;
	MpAXBDrvType : STRUCT (*Drive configuration*)
		MechanicalElements : MpAXBDrvMechElmType; (*Parameter of hardware elements situated between motor encoder and load which influence the scaling*)
		Controller : MpAXBDrvCtrlType; (*Axis controller parameters*)
		Homing : MpAXBDrvHomeType; (*Homing mode and parameters which can be used within the application program as pre-configured setting*)
		StopReaction : MpAXBDrvStopReacType; (*Reactions of the axis in case of certain stop conditions*)
		MovementErrorLimits : MpAXBDrvMovementErrorLimitsType; (*Limit values that result in a stop reaction when exceeded*)
		JerkFilter : MpAXBDrvJerkFilterType; (*Jerk filter*)
		DigitalInputs : MpAXBDrvDigInType; (*Various digital input functionalities e.g. like homing switch or triggers*)
	END_STRUCT;
	MpAxisBasicConfigType : STRUCT (*General purpose datatype*)
		Axis : MpAXBAxType; (*Axis configuration*)
		Drive : MpAXBDrvType; (*Drive configuration*)
	END_STRUCT;
END_TYPE
```

### VisionGlobal.var
```iecst
VAR
	CmdTriggerImage : BOOL;
	CmdShowImageMappView : BOOL;
	CmdSaveFile : BOOL;
END_VAR
```

### Program Logical/Vision/Axis (IEC)

#### Variables.var
```iecst
VAR
	MpAxisBasic_0 : MpAxisBasic;
	AxisPar : MpAxisBasicParType;
END_VAR
```

#### Main.st
```iecst
PROGRAM _INIT
	// This is a simple Task to move an axis. Operation is via the Watch-Window.
	AxisPar.Distance := 20; // [°]
	AxisPar.Velocity := 360; // [°/s]
	AxisPar.Acceleration := 3600; // [°/s^2]
	AxisPar.Deceleration := 3600; // [°/s^2]

END_PROGRAM
PROGRAM _CYCLIC
	// Use the following commands:
	//   MpAxisBasic_0.Power: Switch the axis on
	//   MpAxisBasic_0.Home: Home the axis
	//   MpAxisBasic_0.MoveAdditive: move the arrow on the axis into the field of view
	//   MpAxisBasic_0.MoveVelocity: move the axis continously
	//   MpAxisBasic_0.Update: Activate a new speed after the change OF AxisPar.Velocity

	MpAxisBasic_0.MpLink := ADR(gAxis_1);
	MpAxisBasic_0.Parameters := ADR(AxisPar);
	MpAxisBasic_0.Enable := TRUE;
	MpAxisBasic_0();

END_PROGRAM
```

### Program Logical/Vision/Vi_main (IEC)

#### Main.st
```iecst
PROGRAM _INIT
	// This sample-task triggers a camera with a mappMotion axis
	// In the Vision Application the Trigger Source must be switched to "mapp Axis". In this sample the axis "gAxis_1" is connected to the VisionApplication
	// Usage:
	//   Activate the camera with CmdTriggerImage
	//   Use ViBaseAxisBasedAcquisition_0.AcquisitionParameters.AcquisitionPositions[x] to make one or more trigger points
	//   After the change of Parameters use ViBaseAxisBasedAcquisition_0.Update

	VisionCtrl.Parameters.SetFocus := 6000; // [10µm]
	VisionCtrl.Parameters.ExposureTime := 60; // [µs]
	VisionCtrl.Parameters.FlashColor := 1; // red
	VisionCtrl.Parameters.FlashSegment := 15; // 15 = all Segments
	VisionCtrl.Parameters.EnableVF := TRUE; // Enables the Vision Function (here matching)
END_PROGRAM
PROGRAM _CYCLIC
	// Trigger the camera with the axis
	ViBaseAxisBasedAcquisition_0.Enable := CmdTriggerImage;
	ViBaseAxisBasedAcquisition_0.MpLink := ADR(VCMyCam); // Reference to the camera (vision component), not the axis. The axis is linked in the vision application settings to the camera.
	// ViBaseAxisBasedAcquisition_0.AcquisitionParameters.AcquisitionPositions[0] := 0; // Set the trigger-positions via Watch
	ViBaseAxisBasedAcquisition_0.AcquisitionParameters.Period := 360;
	ViBaseAxisBasedAcquisition_0();

	// Load the image from the camera (task Vi_Image --> CmdShowImageMappView) when the image is ready
	IF VisionCtrl.Status.CompletedAcquisitionCnt <> CompletedAcquisitionCntOld THEN
		CompletedAcquisitionCntOld := VisionCtrl.Status.CompletedAcquisitionCnt;
		CmdShowImageMappView := TRUE;
	END_IF

END_PROGRAM
```

### Program Logical/Vision/Vi_image (IEC)

#### Variables.var
```iecst
VAR CONSTANT
	MAX_IMAGE_SIZE : UDINT := 5320000; (*Details for the calculation of the size see in the INIT*)
	MAX_ENCODED_SIZE : UDINT := 7078000; (*Details for the calculation of the size see in the INIT*)
	MAX_SVG_SIZE : UDINT := 7080000; (*Details for the calculation of the size see in the INIT*)
	IMG_PIXEL_WIDTH : UDINT := 1280; (*See camera documentation*)
	IMG_PIXEL_HEIGHT : UDINT := 1024; (*See camera documentation*)
END_VAR
(**)
VAR
	BufferForBinaryImageData : ARRAY[0..MAX_IMAGE_SIZE] OF USINT; (*Buffer for the raw img-data (bmp or jpg)*)
	BufferForBase64EncodedImageData : ARRAY[0..MAX_ENCODED_SIZE] OF USINT; (*Buffer for t*)
	BufferForSvgCameraImage : STRING[MAX_SVG_SIZE];
	Step : INT;
	ViBaseGetImage_0 : ViBaseGetImage;
	httpEncodeBase64_0 : httpEncodeBase64;
	Status : DINT;
	tmpStr : STRING[80];
END_VAR
(**)
(*File-Handling*)
VAR
	FileDelete_0 : FileDelete;
	FileCreate_0 : FileCreate;
	FileWrite_0 : FileWrite;
	FileClose_0 : FileClose;
END_VAR
```

#### Main.st
```iecst
PROGRAM _INIT
	// This sample-task loads the image from a camera and shows it on a Paper-Widget in mappView
	// A sample with much more functions can also be found here (branch "basic"): https://github.com/br-automation-com/mappVision-Demo/blob/basic/Logical/Vision/Vi_image/Main.st

	// Calculation of buffer-sizes
	// Max image size: 5MP sensor resolution is 2592x2048 Pixel --> 5.308.416 raw Pixels + ~10.000 Byte Overhead --> 5.320.000 Bytes
	// Base 64 is alwas 1/3 bigger: 7.078.000 Bytes
	// The SVG Header is again bigger --> 7.080.000 Bytes
	// Notes:
		// Linesensor: The image could be bigger, depending on used number of lines
		// A jpg-image is compressed, so the buffer can be much smaller. See AS Help.
		// The here saved image with default values (1,3MP, jpg with 80% quality) needs about 350.000 Bytes (0,35 MB)

	// Note: Adapt the constants "IMG_PIXEL_WIDTH/HEIGHT" to the cameras resolution
END_PROGRAM
PROGRAM _CYCLIC
	CASE Step OF

		0: // Wait
			IF CmdShowImageMappView THEN
				CmdShowImageMappView := FALSE;
				ViBaseGetImage_0(Execute := FALSE);
				httpEncodeBase64_0(enable := FALSE);
				// Delete buffers, because of the compressed image (jpg) could be smaller than the last loaded image
				brsmemset(ADR(BufferForBinaryImageData), 0, SIZEOF(BufferForBinaryImageData));
				brsmemset(ADR(BufferForBase64EncodedImageData), 0, SIZEOF(BufferForBase64EncodedImageData));
				Step := 10;
			ELSIF CmdSaveFile THEN
				CmdSaveFile := FALSE;
				Step := 20;
			END_IF

		// Load image, convert to base 64 and generate svg-data for mappView or save as file
		10:  // Load image from camera into variable (internal buffer)
			ViBaseGetImage_0.MpLink := ADR(VCMyCam);
			ViBaseGetImage_0.Execute := TRUE;
			ViBaseGetImage_0.Type := viBASE_IMAGE_TYPE_JPG; // For mappView the compressed jpg is besser for reduced image size
			ViBaseGetImage_0.QualityLevel := 80; // Image is still very good for mappView, but the size is reduced by about 70%
			ViBaseGetImage_0.Timeout := T#5s;
			ViBaseGetImage_0.Buffer := ADR(BufferForBinaryImageData);
			ViBaseGetImage_0.BufferSize := SIZEOF(BufferForBinaryImageData);
			ViBaseGetImage_0();
			IF ViBaseGetImage_0.Done THEN
					Step := 11;
			ELSIF ViBaseGetImage_0.Error THEN
				Status := ViBaseGetImage_0.StatusID;
				IF ViBaseGetImage_0.StatusID = viBASE_ERR_NO_IMG_AVAILABLE THEN // No image --> could happen after startup before first trigger.
					Step := 0;
				ELSE
					Status := ViBaseGetImage_0.StatusID;
					Step := 100;
				END_IF
			END_IF
		11: // Transform image from binary-data to ASCII-data for SVG
			httpEncodeBase64_0.enable := TRUE;
			httpEncodeBase64_0.pSrc := ADR(BufferForBinaryImageData);
			httpEncodeBase64_0.srcLen := ViBaseGetImage_0.BufferLen; // Use the exact length of the image, not the whole buffer
			httpEncodeBase64_0.pDest := ADR(BufferForBase64EncodedImageData);
			httpEncodeBase64_0.destSize := SIZEOF(BufferForBase64EncodedImageData);
			httpEncodeBase64_0();
			IF httpEncodeBase64_0.status = 0 THEN
				Step := 12;
			ELSIF httpEncodeBase64_0.status <> ERR_FUB_BUSY THEN
				Status := httpEncodeBase64_0.status;
				Step := 100;
			END_IF
		12:	// Generate svg-data
			// The svg-data (could also be saved as a file) contains some header and other information.
			// This data will be created as one big string where the image (as base64) is embedded.
			// See also here: https://help.br-automation.com/#/en/4/visualization%2Fmappview%2Fwidgets%2Fdrawing%2Fpaper%2Fkonzept.html
			brsmemset(ADR(BufferForSvgCameraImage), 0, SIZEOF(BufferForSvgCameraImage));
			BufferForSvgCameraImage := '<svg xmlns="http://www.w3.org/2000/svg" width="1280px" height="1024px" viewBox="0 0 ';
			brsitoa(IMG_PIXEL_WIDTH, ADR(tmpStr));
			brsstrcat(ADR(BufferForSvgCameraImage), ADR(tmpStr));
			brsstrcat(ADR(BufferForSvgCameraImage), ADR(' '));
			brsitoa(IMG_PIXEL_HEIGHT, ADR(tmpStr));
			brsstrcat(ADR(BufferForSvgCameraImage), ADR(tmpStr));
			brsstrcat(ADR(BufferForSvgCameraImage), ADR('" xmlns:xlink="http://www.w3.org/1999/xlink"><image xlink:href="data:image/'));
			brsstrcat(ADR(BufferForSvgCameraImage), ADR('jpeg'));
			brsstrcat(ADR(BufferForSvgCameraImage), ADR(';base64,'));
			brsstrcat(ADR(BufferForSvgCameraImage), ADR(BufferForBase64EncodedImageData));
			brsstrcat(ADR(BufferForSvgCameraImage), ADR('"/>'));
			brsstrcat(ADR(BufferForSvgCameraImage), ADR('</svg>'));
			Step := 0;

		// Save svg or jpg file, also bmp is possible
		20:
			FileDelete_0.enable := TRUE;
			FileDelete_0.pDevice := ADR('CF');
			FileDelete_0.pName := ADR('Image.jpg'); // Choose: Save the jpg-file
			//FileDelete_0.pName := ADR('Image.svg'); // Choose: Save the svg-file
			FileDelete_0();
			IF FileDelete_0.status = 0 OR FileDelete_0.status = fiERR_FILE_NOT_FOUND THEN
				Step := 21;
			ELSIF FileDelete_0.status <> ERR_FUB_BUSY THEN
				Status := FileDelete_0.status;
				Step := 100;
			END_IF
		21:
			FileCreate_0.enable := TRUE;
			FileCreate_0.pDevice := FileDelete_0.pDevice;
			FileCreate_0.pFile := FileDelete_0.pName;
			FileCreate_0();
			IF FileCreate_0.status = 0 THEN
				Step := 22;
			ELSIF FileCreate_0.status <> ERR_FUB_BUSY THEN
				Status := FileCreate_0.status;
				Step := 100;
			END_IF
		22:
			FileWrite_0.enable := TRUE;
			FileWrite_0.ident := FileCreate_0.ident;
			FileWrite_0.pSrc := ADR(BufferForBinaryImageData); // Choose: Save the jpg-file
			FileWrite_0.len := ViBaseGetImage_0.BufferLen; // Choose: Save the jpg-file
			//FileWrite_0.pSrc := ADR(BufferForSvgCameraImage); // Choose: Save the svg-file
			//FileWrite_0.len := brsstrlen(ADR(BufferForSvgCameraImage)); // Choose: Save the scg-file
			FileWrite_0();
			IF FileWrite_0.status = 0 THEN
				Step := 23;
			ELSIF FileWrite_0.status <> ERR_FUB_BUSY THEN
				Status := FileWrite_0.status;
				Step := 100;
			END_IF
		23:
			FileClose_0.enable := TRUE;
			FileClose_0.ident := FileCreate_0.ident;
			FileClose_0();
			IF FileClose_0.status = 0 THEN
				Step := 0;
			ELSIF FileClose_0.status <> ERR_FUB_BUSY THEN
				Status := FileClose_0.status;
				Step := 0;
			END_IF

		100: // Error
			// ToDo: Implement some errorhandling here
	END_CASE
END_PROGRAM
```

- Visualisation Logical/mappView (not shown)
